Staubli VAL3: onStart.pgx

program onStart()
  local num i
  local num l_nResult
  local string l_sPath
  local string l_sMessage
begin
  // language
  //
  call language2:getLanguage(l_sPath)
  if l_sPath!=language2:libPath()+"/"+saveData:language
    // set language
    call language2:setLanguage(language2:libPath()+"/"+saveData:language)
  endIf
  // logMsg
  logMsg("[KERNEL] INTERFACE:PAGE VIEW ALL PALLET")
  // reset the Key pressure
  call use:nullKey(nKey)
  call language:message(l_sMessage,19)
  call use:timerDialog(l_sMessage,0)
  // make the max_size of all
  call makeMaxSizeList(l_nResult)
  if l_nResult==0
    //
    call buildList()
    // build the page
    call refreshStatic()
    // define the list
  else
    call language:message(l_sMessage,-7)
    popUpMsg(l_sMessage+" ; "+toString("",l_nResult))
    logMsg("[KERNEL] INTERFACE:ERROR LOADING VIEW PALLET ERROR CODE "+toString("",l_nResult))
  endIf
end
